INTERFACE I_DeferredRpcResponse

METHOD PUBLIC Build : I_ResponseBuilder
VAR_INPUT
END_VAR
END_METHOD

METHOD PUBLIC Reject
VAR_INPUT
	Message : T_MAXSTRING;
END_VAR
END_METHOD

END_INTERFACE

(* stored: Version 1.1.0.1, ProductVersion 3.1.4024.12
   Itf I_DeferredRpcResponse: Id {5ec4868c-976d-405e-84ca-4dd50f0ee2cc}
   Method Build: Id {8927ca37-0e43-4650-a6e3-99a3e977a571}
   Method Reject: Id {b5578681-e311-4557-96af-e76ff958a801} *)
